FUNCTION F_UpdateEventTimeStamp 
VAR_INPUT
	stEvent : REFERENCE TO ST_Event;
END_VAR
VAR
	stFileTime : T_FileTime;
	fbSystemTime   : GETSYSTEMTIME;
END_VAR

fbSystemTime( timeLoDW=>stFileTime.dwLowDateTime, timeHiDW=>stFileTime.dwHighDateTime );
stevent.dtTimeStamp := FILETIME_TO_DT( stFileTime);

END_FUNCTION

(* stored: Version 1.1.0.1, ProductVersion 3.1.4024.16
   POU F_UpdateEventTimeStamp: Id {400e0e5a-7023-4f23-a694-d7ca25d5495e}, SpecialFunc None *)
